KUKA KRL program: chk_w3_grp6_clo.src, chk_w3_grp6_clo.dat

--- chk_w3_grp6_clo.src ---
&ACCESS RV2
&REL 7
&COMMENT Check grampos Z2 Accelo fechado
&PARAM TEMPLATE = C:\KRC\Roboter\Template\vorgabe
&PARAM EDITMASK = *
DEF chk_w3_grp6_clo( )
;FOLD ; Programa de verificacao de grampos Z2 fechado;%{PE}%R 4.1.16,%MKUKATPBASIS,%CCOMMENT,%VNORMAL,%P 2:Programa de verificacao de grampos Z2 fechado
;ENDFOLD
;FOLD ; Modelo Accelo;%{PE}%R 4.1.16,%MKUKATPBASIS,%CCOMMENT,%VNORMAL,%P 2:Modelo Accelo
;ENDFOLD

$TIMER[10] = 0
$TIMER_STOP[10] = FALSE

;FOLD WAIT FOR ( NOT IN 39 'GRAMPO Z2.1 RECUADO ACCELO TRASEIRO' );%{PE}%R 8.2.24,%MKUKATPBASIS,%CEXT_WAIT_FOR,%VEXT_WAIT_FOR,%P 2:, 4:NOT, 5:$IN, 6:39, 7:GRAMPO Z2.1 RECUADO ACCELO TRASEIRO, 9:
WAIT FOR  (  NOT $IN[39] )
;ENDFOLD
;FOLD WAIT FOR ( NOT IN 57 'Z2.2 - Grampo Recuado - Accelo TRASEIRO' );%{PE}%R 8.2.24,%MKUKATPBASIS,%CEXT_WAIT_FOR,%VEXT_WAIT_FOR,%P 2:, 4:NOT, 5:$IN, 6:57, 7:Z2.2 - Grampo Recuado - Accelo TRASEIRO, 9:
WAIT FOR  (  NOT $IN[57] )
;ENDFOLD
;FOLD WAIT FOR ( IN 40 'GRAMPO Z2.1 AVANCADO ACCELO TRASEIRO' );%{PE}%R 8.2.24,%MKUKATPBASIS,%CEXT_WAIT_FOR,%VEXT_WAIT_FOR,%P 2:, 4:, 5:$IN, 6:40, 7:GRAMPO Z2.1 AVANCADO ACCELO TRASEIRO, 9:
WAIT FOR  ( $IN[40] )
;ENDFOLD
;FOLD WAIT FOR ( IN 58 'Z2.2 - Grampo Avançado - Accelo TRASEIRO' );%{PE}%R 8.2.24,%MKUKATPBASIS,%CEXT_WAIT_FOR,%VEXT_WAIT_FOR,%P 2:, 4:, 5:$IN, 6:58, 7:Z2.2 - Grampo Avançado - Accelo TRASEIRO, 9:
WAIT FOR  ( $IN[58] )
;ENDFOLD

$TIMER_STOP[10] = TRUE
$TIMER[10] = 0

END

--- chk_w3_grp6_clo.dat ---
&ACCESS RV2
&REL 7
&COMMENT Check grampos Z2 Accelo fechado
&PARAM TEMPLATE = C:\KRC\Roboter\Template\vorgabe
&PARAM EDITMASK = *
DEFDAT chk_w3_grp6_clo
;FOLD EXTERNAL DECLARATIONS;%{PE}%V3.2.0,%MKUKATPBASIS,%CEXT,%VCOMMON,%P
;FOLD BAS EXT;%{PE}%V3.2.0,%MKUKATPBASIS,%CEXT,%VEXT,%P
EXT  BAS (BAS_COMMAND  :IN,REAL  :IN )
DECL INT SUCCESS
;ENDFOLD
;FOLD GRIPPER EXT;%{E}%V3.2.0,%MKUKATPGRIPPER,%CEXT,%VEXT,%P
EXT  H50 (INT:IN, INT:IN ,INT:IN ,GRP_TYP:IN)
;ENDFOLD
;FOLD SPOT EXT;%{E}%V3.2.0,%MKUKATPSPOT,%CEXT,%VEXT,%P
EXT  USERSPOT (S_COMMAND  :IN, SPOT_TYPE:IN)
;ENDFOLD
;FOLD USER EXT;%{E}%V3.2.0,%MKUKATPUSER,%CEXT,%VEXT,%P
;Make here your modifications
;ENDFOLD
;ENDFOLD

ENDDAT
